// TwinCAT 3 PLC project PLC
// ProgramVersion: 3.1.4024.0
// libraries:
//   Tc2_Standard, * (Beckhoff Automation GmbH)
//   Tc2_System, * (Beckhoff Automation GmbH)
//   Tc3_Module, * (Beckhoff Automation GmbH)
// project tree:
//   DUTs/ DUT.TcDUT
//   GVLs/ GENERAL.TcGVL
//   / PlcTask.TcTTO
//   POUs/ MAIN.TcPOU, Math.TcPOU
// real-time tasks:
//   TASK PlcTask: cycle T#10ms, priority 20, ADS port 350
// I/O:
//   DEVICE Device 1 (EtherCAT), AmsNetId 5.57.24.62.2.1
//     Term 1 (EK1200) [EK1200-5000 EtherCAT Power supply (2A E-Bus)]
//       Term 2 (EL1918) [EL1918, 8Ch. Safety Input 24V, TwinSAFE]
//         modules: Module 1 (FSOE), Module 2 (FSLOGIC)
//       Term 3 (EL2904) [EL2904, 4 Ch. Safety Output 24V, 0.5A, TwinSAFE]
//         modules: Module 1 (FSOES), Module 2 (DO)
//       Term 4 (EL9011) [EL9011 End Terminal]
//   DEVICE Device 4 (COM Port)

CONFIGURATION PLC
    RESOURCE PLC ON TwinCAT3
        TASK PlcTask(INTERVAL := T#10ms, PRIORITY := 20);
        PROGRAM MAIN WITH PlcTask : MAIN;
    END_RESOURCE
END_CONFIGURATION

// ---- DUTs/DUT.TcDUT
TYPE DUT :
UNION
	

bit1	: BOOL;
bit2	: BOOL;
bit3	: BOOL;
bit4	: BOOL;

byte1	: BYTE;



END_UNION
END_TYPE

// ---- GVLs/GENERAL.TcGVL
{attribute 'qualified_only'}
VAR_GLOBAL
	
//Input BOOLS
bDummySw1		:		BOOL;
bDummySw2		:		BOOL;
bDummySw3		: 		BOOL;
bDummySw4		:		BOOL;
bDummySw5		: 	 	BOOL;

//Output BOOLS
bDummyLt1		:		BOOL;
bDummyLt2		:		BOOL;
bDummyLt3		: 		BOOL;
bDummyLt4		:		BOOL;
bDummyLt5		: 	 	BOOL;

//INTS
iDummy1			:		INT;
iDummy2			:		INT;
iDummy3			:		INT;
iDummy4			:		INT;
iDummy5			:		INT;

//REALS
rDummy1			:		REAL;
rDummy2			:		REAL;
rDummy3			:		REAL;
rDummy4			:		REAL;
rDummy5			:		REAL;

//STRINGS
sDummy1			:		STRING;
sDummy2			:		STRING;
sDummy3			:		STRING;
sDummy4			:		STRING;
sDummy5			:		STRING;

END_VAR

// ---- POUs/MAIN.TcPOU
PROGRAM MAIN
VAR
	
calculator		:	Math;
result			:	INT;
unionTest		:	DUT;
byte1			:	BYTE;
int1			:	INT;

END_VAR



calculator.addition(150, 50);

result := calculator.result;

byte1.0 := TRUE;
byte1.1 := TRUE;
byte1.2 := FALSE;
byte1.3 := TRUE;


int1 := BYTE_TO_INT(byte1);

END_PROGRAM

// ---- POUs/Math.TcPOU
FUNCTION_BLOCK Math
VAR_INPUT
	
END_VAR
VAR_OUTPUT
	
result		:	INT;

END_VAR
VAR
END_VAR

METHOD addition : INT
VAR_INPUT
	
input1		:	INT;
input2		:	INT;


END_VAR


result := input1 + input2;
END_METHOD

END_FUNCTION_BLOCK
